% RSLogix 500 project No ONS Solution.RSS, saved by version 8.10.00.18 %
PROJECT "UNTITLED"    % processor: MicroLogix 1500 %

PROGRAM FILES
  LAD 2   3 rungs

DATA FILES
  O0 OUTPUT  4 elements
  I1 INPUT  4 elements
  S2 STATUS  66 elements
  B3 BINARY  4 elements
  T4 TIMER  5 elements
  C5 COUNTER  2 elements
  R6 CONTROL  1 elements
  N7 INTEGER  2 elements
  F8 FLOAT  1 elements

LADDER 2
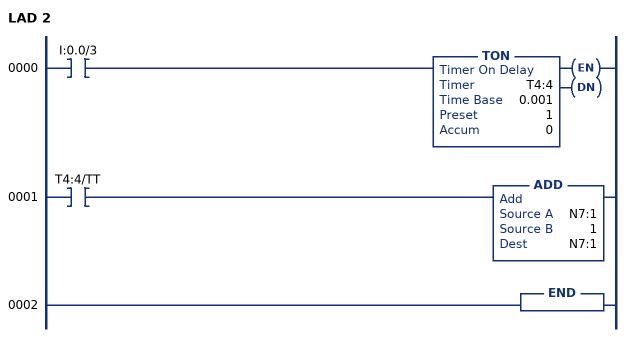
% Rung: 0 %
SOR XIC I:0.0/3 TON T4:4 0.001 1 0 EOR
% Rung: 1 %
SOR XIC T4:4/TT ADD N7:1 1 N7:1 EOR
% Rung: 2 %
SOR END EOR

DATA TABLE (non-zero values as saved)
DATA T4
% .PRE .ACC %
% T4:0 % 50 50
% T4:2 % 1 0
% T4:3 % 100 0
% T4:4 % 1 0
DATA C5
% .PRE .ACC %
% C5:1 % 2 0
